INTERFACE I_InterfaceDatatype_ITcVnBidirectionalIterator EXTENDS I_InterfaceDatatype

PROPERTY PUBLIC Value : REFERENCE TO ITcVnBidirectionalIterator
GET
END_GET
END_PROPERTY

END_INTERFACE

(* stored: Version 1.1.0.1, ProductVersion 3.1.4026.13
   Itf I_InterfaceDatatype_ITcVnBidirectionalIterator: Id {5ba8bb7f-2608-005e-2f67-f11e012d19bc}
   Property Value: Id {db6207b2-e42e-0ca5-0d6f-059d740ff8ed}
   Get Get: Id {e69ebfb1-1e63-0063-3084-40341afb7abc} *)
